TYPE ST_ComIn_ExportStation :
STRUCT
		Enable : BOOL;
		CMD_status: INT;
		StationName:	STRING(30);

END_STRUCT
END_TYPE

(* stored: Version 1.1.0.1
   DUT ST_ComIn_ExportStation: Id {fb89b242-ed00-417e-a233-59a95367b420} *)
